PROGRAM SlitProg
VAR_INPUT
    mySlit : FB_SlitPair_ISIS;

END_VAR

(*SETUP INSTRUCTIONS
    All Axes:
        Allow motion commands to external setpoint axis := FALSE;

    Virtual axes:
        Dynamics of virtual axes must be configured considering coupled mechanicals (e.g. don't set velocities your real axes can't achieve)
*)
mySlit.nIdPositiveAxis := 1;
mySlit.nIdNegativeAxis := 2;
mySlit.nIdGapSizeAxis := 3;
mySlit.nIdGapCentreAxis :=4;
mySlit.bEnable := TRUE;
mySlit();

END_PROGRAM

(* stored: Version 1.1.0.1, ProductVersion 3.1.4024.11
   POU SlitProg: Id {75eb691c-ab1d-43c0-bb0b-1049c83813c7}, SpecialFunc None *)
